// TIA Portal V18 export
DATA_BLOCK "Test_DB"   // DB1
{ S7_Optimized_Access := 'TRUE' }
// stored: MemoryReserve 100
   VAR
      "counter" : UDInt;   // Dilly dally
      test : Bool;
   END_VAR
BEGIN
END_DATA_BLOCK
